RoboDK station: 2D_Curve_V4.rdk

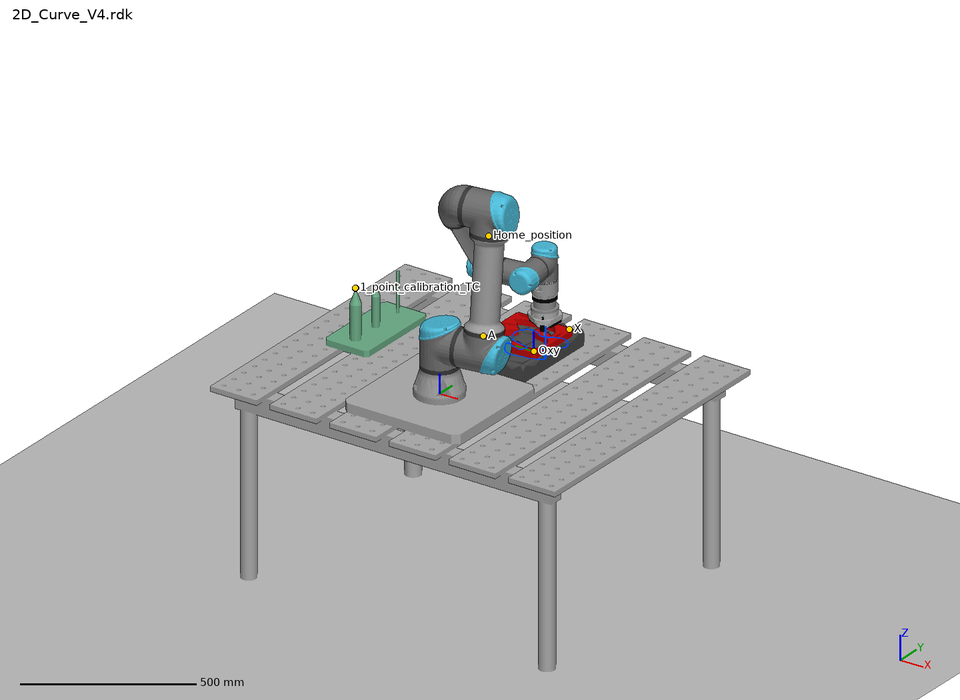
[picture v0: the station drawn from its stored meshes, robots at their saved joint values, targets as dots, program paths as lines]
Station 2D_Curve_V4 (saved by RoboDK 5.6.0). Poses are relative to the parent item; angles as X-Y-Z fixed-axis rotations.
  - frame UR5e Base at (0, 0, 30) mm
    - target Home_position (joint target) at (-5.69, 249.98, 396.72) mm, rotated rx 177.73 ry -1.24 rz 128.57 deg; joints [126, -50.97, -108.8, -108.89, 87.79, -92.57] of UR5e
    - robot UR5e: 6 axes, payload 5 kg, reach 850 mm, repeatability 0.03 mm, weight 18.4 kg
        modified DH rows (alpha deg, a mm, theta deg, d mm): 0, 0, 0, 162.5; 90, 0, 180, 0; 0, 425, 0, 0; 0, 392.25, 0, 133.3; -90, 0, 0, 99.7; 90, 0, 180, 99.6
        joint limits [-360, -360, -360, -360, -360, -360] to [360, 360, 360, 360, 360, 360]; home [0, -90, -90, 0, 90, 0]; saved at [97.663, -96.865, -135.426, -37.71, 90, -172.337]
      - tool Gripper, TCP at (0.02, 0, 134.54) mm, size 93 x 134.6 x 99.8 mm, geometry from UR5e
    - target 1_point_calibration_TCP (joint target) at (-409.67, 170.05, 150.97) mm, rotated rx 177.6 ry 0.93 rz 178.1 deg; joints [-38.669, -91.571, 122.852, -121.97, -92.476, -126.799] of UR5e
    - target 2_point_calibration_TCP (joint target) at (-408.91, 169.63, 151.41) mm, rotated rx 176.95 ry 38.31 rz 176.24 deg; joints [-30.05, -72.145, 98.835, -82.548, -108.779, -111.538] of UR5e
    - target 3_point_calibration_TCP (joint target) at (-409.42, 169.94, 149.48) mm, rotated rx 126.21 ry 38.31 rz 176.24 deg; joints [-13.766, -74.205, 117.825, -108.191, -149.114, -105.406] of UR5e
    - target 4_point_calibration_TCP (joint target) at (-410.09, 169.84, 150.24) mm, rotated rx 173.91 ry -42.23 rz -175.16 deg; joints [-58.732, -99.019, 150.407, -169.44, -56.548, -142.633] of UR5e
    - target Oxy (Cartesian target) at (109.5, 309, 40) mm, rotated rx 180 ry 0 rz 179.32 deg; joints [-265.525, -84.814, -147.79, -37.397, 90, -174.847] of UR5e
    - target X (Cartesian target) at (109.5, 484, 40) mm, rotated rx 180 ry 0 rz 179.32 deg; joints [-267.168, -106.505, -122.454, -41.041, 90, -176.49] of UR5e
    - target A (Cartesian target) at (-65.5, 309, 40) mm, rotated rx 180 ry 0 rz 179.32 deg; joints [-233.073, -82.735, -149.468, -37.797, 90, -142.395] of UR5e
  - object Floor at (-10, -160, -610) mm, size 3000 x 3000 x 0 mm, geometry from Pod.stl
  - object Table at (0, 200, 0) mm, size 1193.8 x 965.2 x 609.6 mm, geometry from Stol.stl
  - object Postolje_UR5e at (0, 0, 0) mm, rotated rx 90 ry 0 rz 0 deg, size 400 x 30 x 400 mm, geometry from Postolje_UR5e.STEP
  - object Sponge at (22, 390, 0) mm, rotated rx 90 ry 0 rz 0 deg, size 200 x 50.9 x 301 mm, geometry from sponge.STEP
  - object Calibration_Gauge at (-410, 270, 0) mm, rotated rx 0 ry 0 rz 90 deg, size 300 x 150 x 180 mm, geometry from kalibracijski_siljak_fiksni_3.stl
  - object 2D_Part at (22, -53, 50) mm, size 195 x 20 x 195 mm, geometry from 2D_Part.STEP
  - frame Frame_Part at (109.5, 309, 70) mm, rotated rx 0 ry 0 rz 90 deg
    - object 2D_Curve at (88, 87.5, -20) mm, rotated rx 0 ry 0 rz 180 deg
  - machining project 2D_Curve settings: rotZ(0) | rotX(0)*rotY(0) | rotz(0) | onStart | onPathStart | onApproach | onPoint | onRetract | onFinish | SetRPM(%1) | SetTool(%1) | Extruder(%1) | default | default | OutOnMov(%1) | OutOffMov(%1) | onPathFinish | M_RunCode(%1)
  - program 2D_Curve (156 instructions, listed below)
  - program Main_Program (7 instructions, listed below)
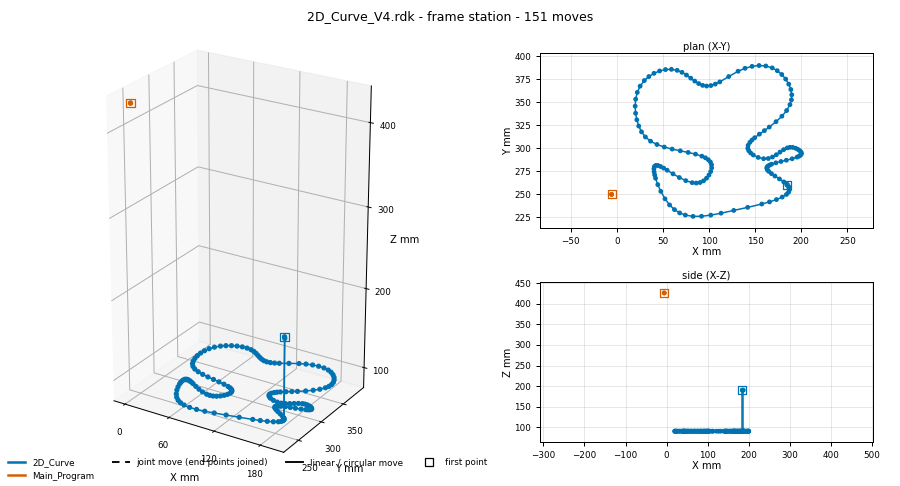
[picture p0: tool path of 2D_Curve_V4.rdk in frame station, 151 of 151 moves have a stored position in this frame; points joined in program order, loops and branches not executed]

--- program 2D_Curve (robot UR5e) ---
  Smooth(1)
  Set speed (1000.0 mm/s)
  Set Ref.: Frame_Part
  Set Tool: Gripper
  Show Gripper
  MoveJ 1 to (-48.55, -75.16, 120) mm, rotated rx 180 ry 0 rz -90 deg; joints [114.083, -89.946, -123.007, -57.047, 90, -155.917]
  MoveL 2 to (-48.55, -75.16, 120) mm, rotated rx 180 ry 0 rz -90 deg; joints [114.083, -89.946, -123.007, -57.047, 90, -155.917]
  MoveL 3 to (-48.55, -75.16, 20) mm, rotated rx -180 ry 0 rz -90 deg; joints [114.083, -101.187, -129.918, -38.895, 90, -155.917]
  MoveL 4 to (-48.55, -75.16, 20) mm, rotated rx -180 ry 0 rz -90 deg; joints [114.083, -101.187, -129.918, -38.895, 90, -155.917]
  Set speed (50.0 mm/s)
  MoveL 5 to (-45.48, -71.51, 20) mm, rotated rx 180 ry 0 rz -90 deg; joints [113.803, -100.785, -130.453, -38.762, 90, -156.197]
  MoveL 6 to (-42.31, -66.87, 20) mm, rotated rx 180 ry 0 rz -90 deg; joints [113.398, -100.36, -131.013, -38.627, 90, -156.602]
  MoveL 7 to (-39.14, -61.96, 20) mm, rotated rx 180 ry 0 rz -90 deg; joints [112.952, -99.933, -131.57, -38.497, 90, -157.048]
  MoveL 8 to (-36.53, -58.19, 20) mm, rotated rx -180 ry 0 rz -90 deg; joints [112.611, -99.589, -132.017, -38.395, 90, -157.389]
  MoveL 9 to (-34.05, -55.19, 20) mm, rotated rx 180 ry 0 rz -90 deg; joints [112.359, -99.267, -132.431, -38.303, 90, -157.641]
  MoveL 10 to (-32.22, -53.67, 20) mm, rotated rx -180 ry 0 rz -90 deg; joints [112.259, -99.035, -132.726, -38.238, 90, -157.741]
  MoveL 11 to (-30.53, -53.12, 20) mm, rotated rx 180 ry 0 rz -90 deg; joints [112.278, -98.828, -132.99, -38.182, 90, -157.722]
  MoveL 12 to (-29.35, -53.47, 20) mm, rotated rx -180 ry 0 rz -90 deg; joints [112.386, -98.691, -133.164, -38.145, 90, -157.614]
  MoveL 13 to (-28.27, -54.5, 20) mm, rotated rx 180 ry 0 rz -90 deg; joints [112.579, -98.57, -133.317, -38.114, 90, -157.421]
  MoveL 14 to (-27.27, -56.12, 20) mm, rotated rx 180 ry 0 rz -90 deg; joints [112.845, -98.465, -133.449, -38.086, 90, -157.155]
  MoveL 15 to (-26.33, -58.24, 20) mm, rotated rx 180 ry 0 rz -90 deg; joints [113.175, -98.374, -133.564, -38.063, 90, -156.825]
  MoveL 16 to (-24.8, -62.98, 20) mm, rotated rx 180 ry 0 rz -90 deg; joints [113.879, -98.242, -133.729, -38.029, 90, -156.121]
  MoveL 17 to (-23.38, -68.52, 20) mm, rotated rx 180 ry 0 rz -90 deg; joints [114.682, -98.139, -133.857, -38.004, 90, -155.318]
  MoveL 18 to (-22, -74.35, 20) mm, rotated rx 180 ry 0 rz -90 deg; joints [115.521, -98.055, -133.962, -37.983, 90, -154.479]
  MoveL 19 to (-20.39, -80.63, 20) mm, rotated rx 180 ry 0 rz -90 deg; joints [116.43, -97.962, -134.078, -37.96, 90, -153.57]
  MoveL 20 to (-18.64, -85.92, 20) mm, rotated rx -180 ry 0 rz -90 deg; joints [117.221, -97.845, -134.223, -37.932, 90, -152.779]
  MoveL 21 to (-17.68, -87.98, 20) mm, rotated rx 180 ry 0 rz -90 deg; joints [117.546, -97.768, -134.319, -37.913, 90, -152.454]
  MoveL 22 to (-16.65, -89.51, 20) mm, rotated rx 180 ry 0 rz -90 deg; joints [117.811, -97.674, -134.436, -37.891, 90, -152.189]
  MoveL 23 to (-15.53, -90.44, 20) mm, rotated rx 180 ry 0 rz -90 deg; joints [118.006, -97.557, -134.58, -37.863, 90, -151.994]
  MoveL 24 to (-14.31, -90.67, 20) mm, rotated rx 180 ry 0 rz -90 deg; joints [118.118, -97.414, -134.756, -37.83, 90, -151.882]
  MoveL 25 to (-12.98, -90.12, 20) mm, rotated rx 180 ry 0 rz -90 deg; joints [118.139, -97.241, -134.967, -37.792, 90, -151.861]
  MoveL 26 to (-11.57, -88.77, 20) mm, rotated rx 180 ry 0 rz -90 deg; joints [118.062, -97.042, -135.21, -37.748, 90, -151.938]
  MoveL 27 to (-10.21, -86.83, 20) mm, rotated rx 180 ry 0 rz -90 deg; joints [117.904, -96.837, -135.459, -37.704, 90, -152.096]
  MoveL 28 to (-9.05, -84.53, 20) mm, rotated rx 180 ry 0 rz -90 deg; joints [117.684, -96.65, -135.685, -37.665, 90, -152.316]
  MoveL 29 to (-8.09, -81.32, 20) mm, rotated rx 180 ry 0 rz -90 deg; joints [117.33, -96.472, -135.899, -37.629, 90, -152.67]
  MoveL 30 to (-7.98, -78.29, 20) mm, rotated rx 180 ry 0 rz -90 deg; joints [116.938, -96.405, -135.98, -37.616, 90, -153.062]
  MoveL 31 to (-8.59, -75.44, 20) mm, rotated rx 180 ry 0 rz -90 deg; joints [116.52, -96.433, -135.946, -37.621, 90, -153.48]
  MoveL 32 to (-10.52, -71.39, 20) mm, rotated rx -180 ry 0 rz -90 deg; joints [115.856, -96.608, -135.735, -37.656, 90, -154.144]
  MoveL 33 to (-13.17, -67.46, 20) mm, rotated rx 180 ry 0 rz -90 deg; joints [115.166, -96.88, -135.407, -37.713, 90, -154.834]
  MoveL 34 to (-16.02, -63.48, 20) mm, rotated rx 180 ry 0 rz -90 deg; joints [114.464, -97.179, -135.043, -37.778, 90, -155.536]
  MoveL 35 to (-18.51, -59.3, 20) mm, rotated rx -180 ry 0 rz -90 deg; joints [113.761, -97.435, -134.729, -37.835, 90, -156.239]
  MoveL 36 to (-20.1, -54.74, 20) mm, rotated rx -180 ry 0 rz -90 deg; joints [113.064, -97.583, -134.548, -37.869, 90, -156.936]
  MoveL 37 to (-20.31, -49.69, 20) mm, rotated rx -180 ry 0 rz -90 deg; joints [112.379, -97.564, -134.571, -37.865, 90, -157.621]
  MoveL 38 to (-18.96, -43.81, 20) mm, rotated rx 180 ry 0 rz -90 deg; joints [111.664, -97.355, -134.827, -37.817, 90, -158.336]
  MoveL 39 to (-16.34, -38.48, 20) mm, rotated rx 180 ry 0 rz -90 deg; joints [111.079, -97.003, -135.258, -37.739, 90, -158.921]
  MoveL 40 to (-14.11, -35.61, 20) mm, rotated rx 180 ry 0 rz -90 deg; joints [110.802, -96.713, -135.609, -37.678, 90, -159.198]
  MoveL 41 to (-11.65, -33.55, 20) mm, rotated rx -180 ry 0 rz -90 deg; joints [110.646, -96.398, -135.987, -37.614, 90, -159.354]
  MoveL 42 to (-9.09, -32.53, 20) mm, rotated rx -180 ry 0 rz -90 deg; joints [110.638, -96.073, -136.375, -37.552, 90, -159.362]
  MoveL 43 to (-5.86, -32.88, 20) mm, rotated rx 180 ry 0 rz -90 deg; joints [110.858, -95.665, -136.857, -37.477, 90, -159.142]
  MoveL 44 to (-2.63, -34.76, 20) mm, rotated rx 180 ry 0 rz -90 deg; joints [111.3, -95.26, -137.331, -37.409, 90, -158.7]
  MoveL 45 to (-0.1, -37.09, 20) mm, rotated rx 180 ry 0 rz -90 deg; joints [111.773, -94.945, -137.696, -37.359, 90, -158.227]
  MoveL 46 to (2.44, -40, 20) mm, rotated rx -180 ry 0 rz -90 deg; joints [112.332, -94.633, -138.055, -37.312, 90, -157.668]
  MoveL 47 to (6.28, -45.1, 20) mm, rotated rx 180 ry 0 rz -90 deg; joints [113.292, -94.168, -138.584, -37.248, 90, -156.708]
  MoveL 48 to (10.12, -50.54, 20) mm, rotated rx 180 ry 0 rz -90 deg; joints [114.312, -93.71, -139.098, -37.192, 90, -155.688]
  MoveL 49 to (13.96, -55.82, 20) mm, rotated rx -180 ry 0 rz -90 deg; joints [115.325, -93.256, -139.602, -37.142, 90, -154.675]
  MoveL 50 to (19.79, -63.14, 20) mm, rotated rx -180 ry 0 rz -90 deg; joints [116.787, -92.57, -140.35, -37.08, 90, -153.213]
  MoveL 51 to (25.73, -69.5, 20) mm, rotated rx 180 ry 0 rz -90 deg; joints [118.15, -91.863, -141.106, -37.031, 90, -151.85]
  MoveL 52 to (31.86, -74.63, 20) mm, rotated rx 180 ry 0 rz -90 deg; joints [119.38, -91.111, -141.893, -36.995, 90, -150.62]
  MoveL 53 to (38.24, -78.24, 20) mm, rotated rx 180 ry 0 rz -90 deg; joints [120.442, -90.29, -142.733, -36.977, 90, -149.558]
  MoveL 54 to (43.49, -79.86, 20) mm, rotated rx 180 ry 0 rz -90 deg; joints [121.139, -89.572, -143.449, -36.979, 90, -148.861]
  MoveL 55 to (48.98, -80.22, 20) mm, rotated rx 180 ry 0 rz -90 deg; joints [121.69, -88.779, -144.222, -36.999, 90, -148.31]
  MoveL 56 to (54.7, -79.23, 20) mm, rotated rx 180 ry 0 rz -90 deg; joints [122.076, -87.898, -145.057, -37.045, 90, -147.924]
  MoveL 57 to (60.47, -76.96, 20) mm, rotated rx 180 ry 0 rz -90 deg; joints [122.284, -86.954, -145.925, -37.122, 90, -147.716]
  MoveL 58 to (66, -73.61, 20) mm, rotated rx 180 ry 0 rz -90 deg; joints [122.307, -85.996, -146.776, -37.227, 90, -147.693]
  MoveL 59 to (70.98, -69.38, 20) mm, rotated rx 180 ry 0 rz -90 deg; joints [122.133, -85.082, -147.564, -37.354, 90, -147.867]
  MoveL 60 to (75.13, -64.46, 20) mm, rotated rx 180 ry 0 rz -90 deg; joints [121.752, -84.275, -148.237, -37.488, 90, -148.248]
  MoveL 61 to (78.15, -59.04, 20) mm, rotated rx 180 ry 0 rz -90 deg; joints [121.159, -83.642, -148.752, -37.606, 90, -148.841]
  MoveL 62 to (80.21, -52.06, 20) mm, rotated rx 180 ry 0 rz -90 deg; joints [120.182, -83.154, -149.14, -37.706, 90, -149.818]
  MoveL 63 to (80.7, -44.72, 20) mm, rotated rx 180 ry 0 rz -90 deg; joints [118.962, -82.958, -149.294, -37.748, 90, -151.038]
  MoveL 64 to (79.81, -37.16, 20) mm, rotated rx 180 ry 0 rz -90 deg; joints [117.552, -83.037, -149.232, -37.731, 90, -152.448]
  MoveL 65 to (77.68, -29.53, 20) mm, rotated rx 180 ry 0 rz -90 deg; joints [116.013, -83.365, -148.973, -37.662, 90, -153.987]
  MoveL 66 to (74.5, -21.99, 20) mm, rotated rx -180 ry 0 rz -90 deg; joints [114.408, -83.904, -148.54, -37.556, 90, -155.592]
  MoveL 67 to (68.74, -11.82, 20) mm, rotated rx 180 ry 0 rz -90 deg; joints [112.167, -84.911, -147.708, -37.381, 90, -157.833]
  MoveL 68 to (62.96, -2.15, 20) mm, rotated rx 180 ry 0 rz -90 deg; joints [110.07, -85.937, -146.828, -37.235, 90, -159.93]
  MoveL 69 to (60.57, 2.73, 20) mm, rotated rx -180 ry 0 rz -90 deg; joints [109.067, -86.375, -146.443, -37.182, 90, -160.933]
  MoveL 70 to (58.97, 7.5, 20) mm, rotated rx 180 ry 0 rz -90 deg; joints [108.141, -86.69, -146.162, -37.148, 90, -161.859]
  MoveL 71 to (58.45, 12.14, 20) mm, rotated rx 180 ry 0 rz -90 deg; joints [107.301, -86.841, -146.026, -37.133, 90, -162.699]
  MoveL 72 to (59.2, 16.48, 20) mm, rotated rx 180 ry 0 rz -90 deg; joints [106.581, -86.797, -146.066, -37.137, 90, -163.419]
  MoveL 73 to (61.12, 20.74, 20) mm, rotated rx -180 ry 0 rz -90 deg; joints [105.928, -86.575, -146.265, -37.16, 90, -164.072]
  MoveL 74 to (63.85, 25.01, 20) mm, rotated rx 180 ry 0 rz -90 deg; joints [105.305, -86.232, -146.569, -37.199, 90, -164.695]
  MoveL 75 to (67.01, 29.34, 20) mm, rotated rx 180 ry 0 rz -90 deg; joints [104.678, -85.828, -146.923, -37.249, 90, -165.322]
  MoveL 76 to (70.36, 34.01, 20) mm, rotated rx -180 ry 0 rz -90 deg; joints [103.984, -85.409, -147.285, -37.306, 90, -166.016]
  MoveL 77 to (73.33, 38.89, 20) mm, rotated rx 180 ry 0 rz -90 deg; joints [103.216, -85.067, -147.576, -37.357, 90, -166.784]
  MoveL 78 to (75.48, 44.07, 20) mm, rotated rx -180 ry 0 rz -90 deg; joints [102.344, -84.882, -147.732, -37.386, 90, -167.656]
  MoveL 79 to (76.57, 50.31, 20) mm, rotated rx 180 ry 0 rz -90 deg; joints [101.221, -84.924, -147.697, -37.379, 90, -168.779]
  MoveL 80 to (76.3, 56.73, 20) mm, rotated rx 180 ry 0 rz -90 deg; joints [100.01, -85.213, -147.452, -37.335, 90, -169.99]
  MoveL 81 to (74.81, 63.11, 20) mm, rotated rx 180 ry 0 rz -90 deg; joints [98.778, -85.711, -147.025, -37.264, 90, -171.222]
  MoveL 82 to (72.24, 69.21, 20) mm, rotated rx 180 ry 0 rz -90 deg; joints [97.585, -86.373, -146.444, -37.182, 90, -172.415]
  MoveL 83 to (68.72, 74.8, 20) mm, rotated rx 180 ry 0 rz -90 deg; joints [96.488, -87.155, -145.742, -37.103, 90, -173.512]
  MoveL 84 to (64.4, 79.67, 20) mm, rotated rx 180 ry 0 rz -90 deg; joints [95.535, -88.013, -144.949, -37.038, 90, -174.465]
  MoveL 85 to (58.34, 84.22, 20) mm, rotated rx 180 ry 0 rz -90 deg; joints [94.641, -89.089, -143.922, -36.989, 90, -175.359]
  MoveL 86 to (51.55, 87.32, 20) mm, rotated rx 180 ry 0 rz -90 deg; joints [94.022, -90.174, -142.85, -36.977, 90, -175.978]
  MoveL 87 to (44.25, 89.07, 20) mm, rotated rx 180 ry 0 rz -90 deg; joints [93.645, -91.242, -141.758, -37, 90, -176.355]
  MoveL 88 to (36.64, 89.64, 20) mm, rotated rx 180 ry 0 rz -90 deg; joints [93.475, -92.273, -140.67, -37.057, 90, -176.525]
  MoveL 89 to (28.94, 89.14, 20) mm, rotated rx 180 ry 0 rz -90 deg; joints [93.48, -93.249, -139.609, -37.142, 90, -176.52]
  MoveL 90 to (21.85, 87.84, 20) mm, rotated rx 180 ry 0 rz -90 deg; joints [93.616, -94.102, -138.658, -37.24, 90, -176.384]
  MoveL 91 to (15.06, 85.76, 20) mm, rotated rx 180 ry 0 rz -90 deg; joints [93.867, -94.878, -137.774, -37.348, 90, -176.133]
  MoveL 92 to (8.78, 82.73, 20) mm, rotated rx 180 ry 0 rz -90 deg; joints [94.26, -95.55, -136.993, -37.457, 90, -175.74]
  MoveL 93 to (3.24, 78.53, 20) mm, rotated rx 180 ry 0 rz -90 deg; joints [94.823, -96.094, -136.351, -37.555, 90, -175.177]
  MoveL 94 to (-1.35, 72.94, 20) mm, rotated rx 180 ry 0 rz -90 deg; joints [95.587, -96.485, -135.883, -37.632, 90, -174.413]
  MoveL 95 to (-4.93, 65.99, 20) mm, rotated rx 180 ry 0 rz -90 deg; joints [96.552, -96.728, -135.591, -37.681, 90, -173.448]
  MoveL 96 to (-7.71, 58.03, 20) mm, rotated rx 180 ry 0 rz -90 deg; joints [97.663, -96.865, -135.426, -37.71, 90, -172.337]
  MoveL 97 to (-9.93, 49.47, 20) mm, rotated rx -180 ry 0 rz -90 deg; joints [98.858, -96.939, -135.335, -37.726, 90, -171.142]
  MoveL 98 to (-11.79, 40.71, 20) mm, rotated rx 180 ry 0 rz -90 deg; joints [100.078, -96.991, -135.272, -37.737, 90, -169.922]
  MoveL 99 to (-13.54, 32.15, 20) mm, rotated rx 180 ry 0 rz -90 deg; joints [101.26, -97.056, -135.193, -37.751, 90, -168.74]
  MoveL 100 to (-15.4, 24.21, 20) mm, rotated rx 180 ry 0 rz -90 deg; joints [102.34, -97.165, -135.06, -37.775, 90, -167.66]
  MoveL 101 to (-17.6, 17.28, 20) mm, rotated rx 180 ry 0 rz -90 deg; joints [103.253, -97.347, -134.838, -37.815, 90, -166.747]
  MoveL 102 to (-19.36, 13.42, 20) mm, rotated rx 180 ry 0 rz -90 deg; joints [103.737, -97.52, -134.625, -37.855, 90, -166.263]
  MoveL 103 to (-21.45, 10.3, 20) mm, rotated rx -180 ry 0 rz -90 deg; joints [104.101, -97.744, -134.349, -37.907, 90, -165.899]
  MoveL 104 to (-23.92, 8.06, 20) mm, rotated rx 180 ry 0 rz -90 deg; joints [104.327, -98.023, -134.002, -37.975, 90, -165.673]
  MoveL 105 to (-26.84, 6.8, 20) mm, rotated rx 180 ry 0 rz -90 deg; joints [104.397, -98.366, -133.573, -38.061, 90, -165.603]
  MoveL 106 to (-30.28, 6.65, 20) mm, rotated rx 180 ry 0 rz -90 deg; joints [104.297, -98.779, -133.053, -38.169, 90, -165.703]
  MoveL 107 to (-34.28, 7.7, 20) mm, rotated rx 180 ry 0 rz -90 deg; joints [104.017, -99.264, -132.434, -38.302, 90, -165.983]
  MoveL 108 to (-38.03, 9.6, 20) mm, rotated rx 180 ry 0 rz -90 deg; joints [103.637, -99.724, -131.842, -38.434, 90, -166.363]
  MoveL 109 to (-41.54, 12.25, 20) mm, rotated rx 180 ry 0 rz -90 deg; joints [103.171, -100.159, -131.276, -38.565, 90, -166.829]
  MoveL 110 to (-44.39, 15.52, 20) mm, rotated rx -180 ry 0 rz -90 deg; joints [102.65, -100.522, -130.8, -38.678, 90, -167.35]
  MoveL 111 to (-46.17, 19.28, 20) mm, rotated rx 180 ry 0 rz -90 deg; joints [102.102, -100.768, -130.475, -38.757, 90, -167.898]
  MoveL 112 to (-46.76, 23.4, 20) mm, rotated rx 180 ry 0 rz -90 deg; joints [101.542, -100.882, -130.324, -38.794, 90, -168.458]
  MoveL 113 to (-46.32, 27.8, 20) mm, rotated rx 180 ry 0 rz -90 deg; joints [100.973, -100.886, -130.319, -38.795, 90, -169.027]
  MoveL 114 to (-44.15, 34.72, 20) mm, rotated rx 180 ry 0 rz -90 deg; joints [100.11, -100.732, -130.523, -38.745, 90, -169.89]
  MoveL 115 to (-40.75, 41.75, 20) mm, rotated rx -180 ry 0 rz -90 deg; joints [99.249, -100.451, -130.894, -38.656, 90, -170.751]
  MoveL 116 to (-36.76, 48.58, 20) mm, rotated rx 180 ry 0 rz -90 deg; joints [98.412, -100.111, -131.338, -38.55, 90, -171.588]
  MoveL 117 to (-32.84, 54.91, 20) mm, rotated rx 180 ry 0 rz -90 deg; joints [97.626, -99.781, -131.768, -38.451, 90, -172.374]
  MoveL 118 to (-30.57, 58.7, 20) mm, rotated rx 180 ry 0 rz -90 deg; joints [97.148, -99.598, -132.004, -38.398, 90, -172.852]
  MoveL 119 to (-28.8, 62.05, 20) mm, rotated rx 180 ry 0 rz -90 deg; joints [96.717, -99.468, -132.172, -38.36, 90, -173.283]
  MoveL 120 to (-27.74, 64.85, 20) mm, rotated rx 180 ry 0 rz -90 deg; joints [96.348, -99.409, -132.247, -38.343, 90, -173.652]
  MoveL 121 to (-27.6, 67.25, 20) mm, rotated rx 180 ry 0 rz -90 deg; joints [96.019, -99.452, -132.193, -38.355, 90, -173.981]
  MoveL 122 to (-28.85, 68.72, 20) mm, rotated rx 180 ry 0 rz -90 deg; joints [95.798, -99.632, -131.96, -38.408, 90, -174.202]
  MoveL 123 to (-31.27, 69.27, 20) mm, rotated rx -180 ry 0 rz -90 deg; joints [95.69, -99.925, -131.581, -38.494, 90, -174.31]
  MoveL 124 to (-34.68, 69.08, 20) mm, rotated rx 180 ry 0 rz -90 deg; joints [95.669, -100.312, -131.075, -38.612, 90, -174.331]
  MoveL 125 to (-37.91, 68.48, 20) mm, rotated rx 180 ry 0 rz -90 deg; joints [95.707, -100.667, -130.609, -38.724, 90, -174.293]
  MoveL 126 to (-41.5, 67.52, 20) mm, rotated rx 180 ry 0 rz -90 deg; joints [95.787, -101.053, -130.097, -38.85, 90, -174.213]
  MoveL 127 to (-48.49, 65.06, 20) mm, rotated rx 180 ry 0 rz -90 deg; joints [96.017, -101.788, -129.112, -39.101, 90, -173.983]
  MoveL 128 to (-55.7, 61.84, 20) mm, rotated rx 180 ry 0 rz -90 deg; joints [96.334, -102.526, -128.106, -39.367, 90, -173.666]
  MoveL 129 to (-63.84, 57.28, 20) mm, rotated rx 180 ry 0 rz -90 deg; joints [96.799, -103.341, -126.982, -39.678, 90, -173.201]
  MoveL 130 to (-70.48, 52.32, 20) mm, rotated rx 180 ry 0 rz -90 deg; joints [97.32, -103.984, -126.082, -39.935, 90, -172.68]
  MoveL 131 to (-75.53, 47.02, 20) mm, rotated rx 180 ry 0 rz -90 deg; joints [97.896, -104.451, -125.421, -40.128, 90, -172.104]
  MoveL 132 to (-79.15, 41.32, 20) mm, rotated rx 180 ry 0 rz -90 deg; joints [98.533, -104.761, -124.98, -40.259, 90, -171.467]
  MoveL 133 to (-81.5, 35.19, 20) mm, rotated rx 180 ry 0 rz -90 deg; joints [99.239, -104.934, -124.733, -40.333, 90, -170.761]
  MoveL 134 to (-82.87, 26.85, 20) mm, rotated rx 180 ry 0 rz -90 deg; joints [100.227, -104.982, -124.663, -40.354, 90, -169.773]
  MoveL 135 to (-82.78, 17.68, 20) mm, rotated rx 180 ry 0 rz -90 deg; joints [101.345, -104.88, -124.81, -40.31, 90, -168.655]
  MoveL 136 to (-81.53, 7.57, 20) mm, rotated rx 180 ry 0 rz -90 deg; joints [102.603, -104.662, -125.122, -40.217, 90, -167.397]
  MoveL 137 to (-79.43, -3.54, 20) mm, rotated rx -180 ry 0 rz -90 deg; joints [104.013, -104.367, -125.541, -40.093, 90, -165.987]
  MoveL 138 to (-76.43, -17.29, 20) mm, rotated rx 180 ry 0 rz -90 deg; joints [105.78, -103.995, -126.066, -39.939, 90, -164.22]
  MoveL 139 to (-73.11, -32.4, 20) mm, rotated rx 180 ry 0 rz -90 deg; joints [107.733, -103.634, -126.573, -39.793, 90, -162.267]
  MoveL 140 to (-69.5, -47.69, 20) mm, rotated rx 180 ry 0 rz -90 deg; joints [109.727, -103.295, -127.046, -39.66, 90, -160.273]
  MoveL 141 to (-67.18, -56.08, 20) mm, rotated rx 180 ry 0 rz -90 deg; joints [110.839, -103.095, -127.323, -39.582, 90, -159.161]
  MoveL 142 to (-64.69, -63.58, 20) mm, rotated rx 180 ry 0 rz -90 deg; joints [111.855, -102.883, -127.615, -39.501, 90, -158.145]
  MoveL 143 to (-62, -69.83, 20) mm, rotated rx -180 ry 0 rz -90 deg; joints [112.736, -102.649, -127.939, -39.413, 90, -157.264]
  MoveL 144 to (-59.08, -74.48, 20) mm, rotated rx 180 ry 0 rz -90 deg; joints [113.441, -102.376, -128.312, -39.312, 90, -156.559]
  MoveL 145 to (-56.69, -76.72, 20) mm, rotated rx -180 ry 0 rz -90 deg; joints [113.834, -102.137, -128.638, -39.225, 90, -156.166]
  MoveL 146 to (-54.15, -77.68, 20) mm, rotated rx 180 ry 0 rz -90 deg; joints [114.085, -101.862, -129.011, -39.127, 90, -155.915]
  MoveL 147 to (-51.44, -77.21, 20) mm, rotated rx -180 ry 0 rz -90 deg; joints [114.175, -101.547, -129.436, -39.017, 90, -155.825]
  Set speed (1000.0 mm/s)
  MoveL 148 to (-51.44, -77.21, 20) mm, rotated rx -180 ry 0 rz -90 deg; joints [114.175, -101.547, -129.436, -39.017, 90, -155.825]
  MoveL 149 to (-51.44, -77.21, 120) mm, rotated rx 180 ry 0 rz -90 deg; joints [114.175, -90.386, -122.565, -57.049, 90, -155.825]

--- program Main_Program (robot UR5e) ---
  Smooth(100)
  Set Tool: Gripper
  Set speed (200.0 mm/s)
  Set Ref.: UR5e Base
  MoveJ (Home_position)
  Call 2D_Curve
  MoveJ (Home_position)
